RoboDK station: Store.rdk

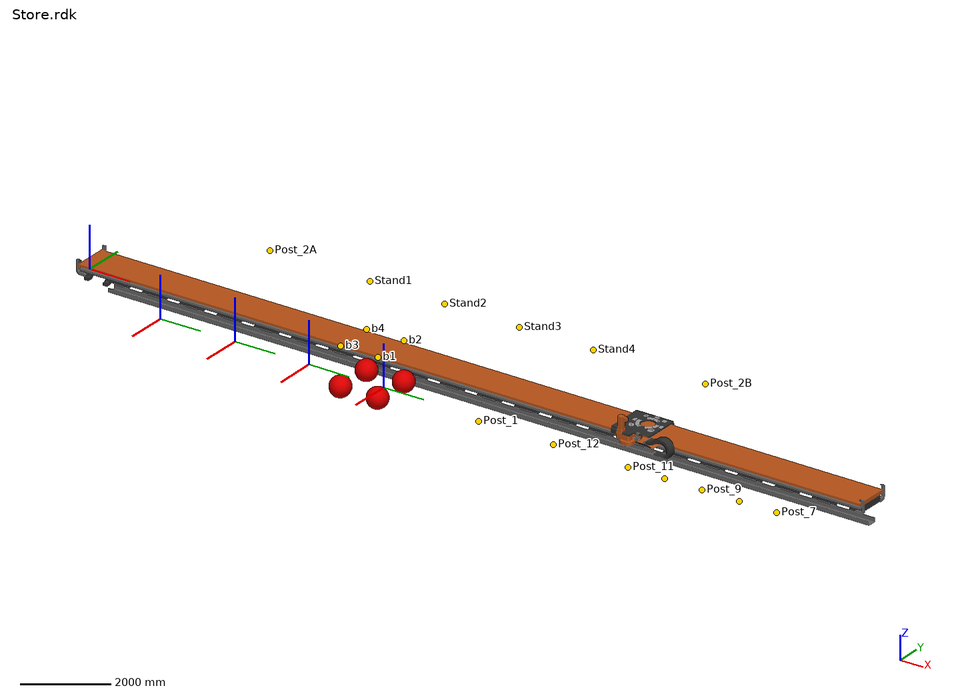
[picture v0: the station drawn from its stored meshes, robots at their saved joint values, targets as dots, program paths as lines]
Station UranStore. Poses are relative to the parent item; angles as X-Y-Z fixed-axis rotations.
  - Python program AddRobots (listed below)
  - Python program SetJobs (listed below)
  - program MainProgram (2 instructions, listed below)
  - frame ABB IRBT 4004 Standard 20m Base at (0, 1000, 0) mm
    - robot Platform: 1 axes, repeatability 0.1 mm
        modified DH rows (alpha deg, a mm, theta deg, d mm): 0, 0, 0, 0 linear
        base shift (645.5, 86.8, 370.5) mm, rotated rx 0 ry 90 rz 0 deg
        joint limits [0] to [20000]; home [0]; saved at [14300]
    - target Post_1 (Cartesian target) at (12000, -2200, 500) mm, rotated rx 180 ry 0 rz 0 deg; joints [-59.361, 68.535, -33.954, 0, -56.046, 59.361, 10000]
    - target Post_2A (Cartesian target) at (3300, 2200, 500) mm, rotated rx -180 ry 0 rz 0 deg; joints [129.557, 74.955, -28.398, 0, -61.602, -129.557, 4400]
    - target Stand1 (Cartesian target) at (6000, 2200, 500) mm, rotated rx 180 ry 0 rz 0 deg; joints [50.299, 75.485, -27.939, 0, -62.061, -50.299, 3600]
    - target Stand2 (Cartesian target) at (8000, 2200, 500) mm, rotated rx 180 ry 0 rz 0 deg; joints [50.299, 75.485, -27.939, 0, -62.061, 309.701, 5600]
    - target Stand3 (Cartesian target) at (10000, 2200, 500) mm, rotated rx 180 ry 0 rz 0 deg; joints [53.661, 66.312, -35.875, 0, -54.125, 306.339, 7800]
    - target Stand4 (Cartesian target) at (12000, 2200, 500) mm, rotated rx 180 ry 0 rz 0 deg; joints [50.299, 75.485, -27.939, 0, -62.061, -50.299, 9600]
    - target b4 (Cartesian target) at (8500, -1500, 1500) mm, rotated rx 180 ry 0 rz 0 deg; joints [-108.972, -1.15, -20.696, 0, -69.304, 108.972, 8400]
    - target b3 (Cartesian target) at (8500, -2500, 1500) mm, rotated rx 180 ry 0 rz 0 deg; joints [-75.801, 68.282, 10.708, 0, -100.708, 75.801, 7200]
    - target b2 (Cartesian target) at (9500, -1500, 1500) mm, rotated rx 180 ry 0 rz 0 deg; joints [-37.681, 53.216, -0.942, 0, -89.058, 37.681, 6800]
    - target b1 (Cartesian target) at (9500, -2500, 1500) mm, rotated rx 180 ry 0 rz 0 deg; joints [-75.801, 68.282, 10.708, 0, -100.708, 75.801, 8200]
    - object Sphere 0.6m 1 at (9500, -1500, 500) mm, rotated rx -180 ry 0 rz -90 deg, size 520.2 x 520.2 x 520.2 mm, geometry from sphere_1m.sld
    - object Sphere 0.6m 2 at (8500, -1500, 500) mm, rotated rx -180 ry 0 rz -90 deg, size 520.2 x 520.2 x 520.2 mm, geometry from sphere_1m.sld
    - object Sphere 0.6m 3 at (8500, -2500, 500) mm, rotated rx -180 ry 0 rz -90 deg, size 520.2 x 520.2 x 520.2 mm, geometry from sphere_1m.sld
    - target Post_2B (Cartesian target) at (15000, 2200, 500) mm, rotated rx -180 ry 0 rz 0 deg; joints [50.299, 75.485, -27.939, 0, -62.061, -50.299, 12600]
    - target Post_7 (Cartesian target) at (20000, -2200, 500) mm, rotated rx -180 ry 0 rz 0 deg; joints [-91.14, 49.966, -49.846, 0, -40.154, 91.14, 19400]
    - target Post_8 (Cartesian target) at (19000, -2200, 500) mm, rotated rx 180 ry 0 rz 0 deg; joints [-59.361, 68.535, -33.954, 0, -56.046, 59.361, 17000]
    - target Post_9 (Cartesian target) at (18000, -2200, 500) mm, rotated rx 180 ry 0 rz 0 deg; joints [-59.361, 68.535, -33.954, 0, -56.046, 59.361, 16000]
    - target Post_10 (Cartesian target) at (17000, -2200, 500) mm, rotated rx 180 ry 0 rz 0 deg; joints [-59.361, 68.535, -33.954, 0, -56.046, 59.361, 15000]
    - target Post_11 (Cartesian target) at (16000, -2200, 500) mm, rotated rx 180 ry 0 rz 0 deg; joints [-59.361, 68.535, -33.954, 0, -56.046, 59.361, 14000]
    - target Post_12 (Cartesian target) at (14000, -2200, 500) mm, rotated rx 180 ry 0 rz 0 deg; joints [-71.74, 55.123, -45.481, 0, -44.519, 71.74, 12600]
    - frame Pallet1 at (10000, -3000, 1100) mm, rotated rx 0 ry 0 rz -90 deg
    - frame Pallet2 at (8000, -3000, 1100) mm, rotated rx 0 ry 0 rz -90 deg
    - frame Pallet3 at (6000, -3000, 1100) mm, rotated rx 0 ry 0 rz -90 deg
    - object Sphere 0.6m 4 at (9500, -2500, 500) mm, rotated rx -180 ry 0 rz -90 deg, size 520.2 x 520.2 x 520.2 mm, geometry from sphere_1m.sld
    - frame Pallet4 at (4000, -3000, 1100) mm, rotated rx 0 ry 0 rz -90 deg

--- Python program AddRobots ---
# Type help("robolink") or help("robodk") for more information
# Press F5 to run the script
# Or visit: http://www.robodk.com/doc/PythonAPI/
# Note: you do not need to keep a copy of this file, your python script is saved with the station
from robolink import *    # API to communicate with RoboDK
from robodk import *      # basic matrix operations
RDK = Robolink()

#robot = RDK.AddFile('C:\projects\Fanuc-M-900iB-700.robot')
robot = RDK.AddFile('Fanuc-M-900iB-700.robot')
#platform = RDK.AddFile('C:\projects\ABB-IRBT-4004-Standard-20m.robot')
platform = RDK.Item('Platform')
robotFrame = RDK.Item('Fanuc M-900iB/700 base')
robotFrame.setParent(platform)
robotFrame.setPose(transl(0,0,930))

robot.AddTool(transl(0,0,400),'Tool')

--- Python program SetJobs ---
# Type help("robolink") or help("robodk") for more information
# Press F5 to run the script
# Or visit: http://www.robodk.com/doc/PythonAPI/
# Note: you do not need to keep a copy of this file, your python script is saved with the station
from robolink import *    # API to communicate with RoboDK
from robodk import *      # basic matrix operations
RDK = Robolink()

#robot = RDK.Item('Fanuc M-900iB/700')
robot = RDK.Item('Platform').Childs()[0].Childs()[0]
robot.setName('Robot')
target1 = RDK.Item('Post_1')
target1.setRobot(robot)
target2a = RDK.Item('Post_2A')
target2a.setRobot(robot)
target2b = RDK.Item('Post_2B')
target2b.setRobot(robot)

target7_12 = []
for i in range(7,13):
    target7_12.append(RDK.Item('Post_'+str(i)))
    target7_12[i-1-6].setRobot(robot)

stands = []
for i in range(1,4+1):
    stands.append(RDK.Item('Stand'+str(i)))
    #print(stands[i-1].Name())
    stands[i-1].setRobot(robot)

pal_bar_count = 4
pal_barrels = []
for i in range(1,pal_bar_count+1):
    pal_barrels.append(RDK.Item('b'+str(i)))
    pal_barrels[i-1].setRobot(robot)
    print(pal_barrels[i-1].Name())

--- program MainProgram (robot Platform) ---
  Call AddRobots
  Call SetJobs
